PROGRAM MAIN
VAR
END_VAR

END_PROGRAM

(* stored: Version 1.1.0.1
   POU MAIN: Id {e88c3478-2b7c-40b0-92b5-a41aea6b8b4e} *)
